// TwinCAT 3 PLC project MAIN
// ProgramVersion: 3.1.4026.24
// libraries:
//   Tc2_Standard, * (Beckhoff Automation GmbH)
//   Tc2_System, * (Beckhoff Automation GmbH)
// project tree:
//   DUTs/ E_AutoStep.TcDUT, E_HostCmdId.TcDUT, E_MachineState.TcDUT, ST_HostCmd.TcDUT, ST_PlcState.TcDUT
//   GVLs/ GVL_HMI.TcGVL
//   / PlcTask.TcTTO
//   POUs/ FB_AutoProcess.TcPOU, FB_HmiInterface.TcPOU, MAIN.TcPOU
// real-time tasks:
//   TASK PlcTask: cycle T#10ms, priority 20, ADS port 350

CONFIGURATION MAIN
    RESOURCE PLC ON TwinCAT3
        TASK PlcTask(INTERVAL := T#10ms, PRIORITY := 20);
        PROGRAM MAIN WITH PlcTask : MAIN;
    END_RESOURCE
END_CONFIGURATION

// ---- DUTs/E_AutoStep.TcDUT
TYPE E_AutoStep :
(
    Idle              := 0,
    CheckReady        := 10,
    TrayFeed          := 20,
    PickProduct       := 30,
    TopVisionAngle    := 40,
    RotateProduct     := 50,
    PlaceToRing       := 60,
    RingToClamp       := 70,
    ClampProduct      := 80,
    CoaxVision        := 90,
    CoaxAdjust        := 100,
    ScrewMove         := 110,
    ScrewTighten      := 120,
    RingReturn        := 130,
    PickBack          := 140,
    PlaceToTray       := 150,
    NextProduct       := 160,
    Finished          := 170,
    Error             := 999
);
END_TYPE

// ---- DUTs/E_HostCmdId.TcDUT
TYPE E_HostCmdId :
(
    None        := 0,
    StartAuto   := 1,
    Pause       := 2,
    ContinueRun := 3,
    Stop        := 4,
    Reset       := 5,
    ClearAlarm  := 6,
    HomeAll     := 7,
    ToManual    := 8,
    ToAuto      := 9,
    ManualAct   := 10
);
END_TYPE

// ---- DUTs/E_MachineState.TcDUT
TYPE E_MachineState :
(
    PowerOnCheck := 0,
    NeedHome     := 10,
    Homing       := 20,
    Standby      := 30,
    AutoRunning  := 40,
    Paused       := 50,
    Stopping     := 60,
    Alarm        := 70,
    Manual       := 80,
    Maintenance  := 90
);
END_TYPE

// ---- DUTs/ST_HostCmd.TcDUT
TYPE ST_HostCmd :
STRUCT
    Heartbeat       : UDINT;        // 上位机心跳
    CmdSeq          : UDINT;        // 命令序号，每发一次命令加 1
    CmdId           : E_HostCmdId;  // 命令编号
    RecipeId        : UINT;         // 配方号
    ManualStationId : UINT;         // 手动工位编号
    ManualActionId  : UINT;         // 手动动作编号
END_STRUCT
END_TYPE

// ---- DUTs/ST_PlcState.TcDUT
TYPE ST_PlcState :
STRUCT
    Heartbeat      : UDINT;           // PLC 心跳
    AckSeq         : UDINT;           // 已响应的命令序号
    MachineState   : E_MachineState;  // 设备总状态
    CurrentStep    : E_AutoStep;      // 当前自动工步
    AlarmCode      : UDINT;           // 当前报警代码

    AutoRunning    : BOOL;            // 自动运行中
    Paused         : BOOL;            // 暂停中
    AxisAllReady   : BOOL;            // 所有轴就绪
    EtherCATReady  : BOOL;            // EtherCAT 正常

    CurrentTray    : UINT;            // 当前料盘编号
    CurrentRow     : UINT;            // 当前行
    CurrentColumn  : UINT;            // 当前列

    GoodCount      : UDINT;           // OK 数量
    NgCount        : UDINT;           // NG 数量
    CycleTimeMs    : LREAL;           // 单件节拍
END_STRUCT
END_TYPE

// ---- GVLs/GVL_HMI.TcGVL
VAR_GLOBAL
    gHostCmd  : ST_HostCmd;   // 上位机写入
    gPlcState : ST_PlcState;  // PLC 返回上位机
END_VAR

// ---- POUs/MAIN.TcPOU
PROGRAM MAIN
VAR
    fbHmiInterface : FB_HmiInterface;
    fbAutoProcess  : FB_AutoProcess;
END_VAR

// 处理上位机命令
fbHmiInterface();

// 自动流程状态机
fbAutoProcess();

END_PROGRAM

// ---- POUs/FB_HmiInterface.TcPOU
FUNCTION_BLOCK FB_HmiInterface
VAR
    lastCmdSeq : UDINT := 0;
END_VAR

GVL_HMI.gPlcState.Heartbeat := GVL_HMI.gPlcState.Heartbeat + 1;

GVL_HMI.gPlcState.AxisAllReady := TRUE;
GVL_HMI.gPlcState.EtherCATReady := TRUE;

IF GVL_HMI.gPlcState.MachineState = 0 THEN
    GVL_HMI.gPlcState.MachineState := 30;
END_IF

IF GVL_HMI.gHostCmd.CmdSeq <> lastCmdSeq THEN

    lastCmdSeq := GVL_HMI.gHostCmd.CmdSeq;

    CASE GVL_HMI.gHostCmd.CmdId OF

        1:
            IF GVL_HMI.gPlcState.MachineState = 30 THEN
                GVL_HMI.gPlcState.MachineState := 40;
                GVL_HMI.gPlcState.AutoRunning := TRUE;
                GVL_HMI.gPlcState.Paused := FALSE;
                GVL_HMI.gPlcState.CurrentStep := 0;
            END_IF

        2:
            IF GVL_HMI.gPlcState.MachineState = 40 THEN
                GVL_HMI.gPlcState.MachineState := 50;
                GVL_HMI.gPlcState.AutoRunning := FALSE;
                GVL_HMI.gPlcState.Paused := TRUE;
            END_IF

        3:
            IF GVL_HMI.gPlcState.MachineState = 50 THEN
                GVL_HMI.gPlcState.MachineState := 40;
                GVL_HMI.gPlcState.AutoRunning := TRUE;
                GVL_HMI.gPlcState.Paused := FALSE;
            END_IF

        4:
            GVL_HMI.gPlcState.MachineState := 30;
            GVL_HMI.gPlcState.AutoRunning := FALSE;
            GVL_HMI.gPlcState.Paused := FALSE;
            GVL_HMI.gPlcState.CurrentStep := 0;

        5:
            GVL_HMI.gPlcState.AlarmCode := 0;
            GVL_HMI.gPlcState.MachineState := 30;
            GVL_HMI.gPlcState.AutoRunning := FALSE;
            GVL_HMI.gPlcState.Paused := FALSE;
            GVL_HMI.gPlcState.CurrentStep := 0;

        6:
            GVL_HMI.gPlcState.AlarmCode := 0;
            IF GVL_HMI.gPlcState.MachineState = 70 THEN
                GVL_HMI.gPlcState.MachineState := 30;
            END_IF

    END_CASE

    GVL_HMI.gPlcState.AckSeq := lastCmdSeq;

END_IF

END_FUNCTION_BLOCK

// ---- POUs/FB_AutoProcess.TcPOU
FUNCTION_BLOCK FB_AutoProcess
VAR
    stepTimer : TON;
    stepDelay : TIME := T#1S;
END_VAR

// 只有自动运行状态才推进流程
IF GVL_HMI.gPlcState.MachineState <> 40 THEN // AutoRunning
    stepTimer(IN := FALSE);
    RETURN;
END_IF

// 每一步延时 1 秒，方便上位机观察工步变化
stepTimer(IN := TRUE, PT := stepDelay);

IF NOT stepTimer.Q THEN
    RETURN;
END_IF

// 定时器到达后复位，准备下一步
stepTimer(IN := FALSE);

CASE GVL_HMI.gPlcState.CurrentStep OF

    0: // Idle
        GVL_HMI.gPlcState.CurrentStep := 10; // CheckReady

    10: // CheckReady
        IF GVL_HMI.gPlcState.AxisAllReady AND GVL_HMI.gPlcState.EtherCATReady THEN
            GVL_HMI.gPlcState.CurrentStep := 20; // TrayFeed
        ELSE
            GVL_HMI.gPlcState.AlarmCode := 1001;
            GVL_HMI.gPlcState.MachineState := 70; // Alarm
        END_IF

    20: // TrayFeed 料盘补给
        GVL_HMI.gPlcState.CurrentStep := 30; // PickProduct

    30: // PickProduct 三轴取料
        GVL_HMI.gPlcState.CurrentStep := 40; // TopVisionAngle

    40: // TopVisionAngle 角度相机识别
        GVL_HMI.gPlcState.CurrentStep := 50; // RotateProduct

    50: // RotateProduct 旋转夹爪校正角度
        GVL_HMI.gPlcState.CurrentStep := 60; // PlaceToRing

    60: // PlaceToRing 放入环形备料位
        GVL_HMI.gPlcState.CurrentStep := 70; // RingToClamp

    70: // RingToClamp 环形区旋转到夹紧位
        GVL_HMI.gPlcState.CurrentStep := 80; // ClampProduct

    80: // ClampProduct 夹紧产品
        GVL_HMI.gPlcState.CurrentStep := 90; // CoaxVision

    90: // CoaxVision 同轴度检测
        GVL_HMI.gPlcState.CurrentStep := 100; // CoaxAdjust

    100: // CoaxAdjust 同轴度调整
        GVL_HMI.gPlcState.CurrentStep := 110; // ScrewMove

    110: // ScrewMove 电批移动
        GVL_HMI.gPlcState.CurrentStep := 120; // ScrewTighten

    120: // ScrewTighten 拧紧螺钉
        GVL_HMI.gPlcState.CurrentStep := 130; // RingReturn

    130: // RingReturn 夹紧位旋回备料位
        GVL_HMI.gPlcState.CurrentStep := 140; // PickBack

    140: // PickBack 三轴取回产品
        GVL_HMI.gPlcState.CurrentStep := 150; // PlaceToTray

    150: // PlaceToTray 放回料盘
        GVL_HMI.gPlcState.GoodCount := GVL_HMI.gPlcState.GoodCount + 1;
        GVL_HMI.gPlcState.CurrentColumn := GVL_HMI.gPlcState.CurrentColumn + 1;
        GVL_HMI.gPlcState.CurrentStep := 160; // NextProduct

    160: // NextProduct 下一个产品
        IF GVL_HMI.gPlcState.CurrentColumn >= 6 THEN
            GVL_HMI.gPlcState.CurrentColumn := 0;
            GVL_HMI.gPlcState.CurrentRow := GVL_HMI.gPlcState.CurrentRow + 1;
        END_IF

        IF GVL_HMI.gPlcState.CurrentRow >= 4 THEN
            GVL_HMI.gPlcState.CurrentRow := 0;
            GVL_HMI.gPlcState.CurrentTray := GVL_HMI.gPlcState.CurrentTray + 1;
        END_IF

        IF GVL_HMI.gPlcState.CurrentTray >= 5 THEN
            GVL_HMI.gPlcState.CurrentStep := 170; // Finished
        ELSE
            GVL_HMI.gPlcState.CurrentStep := 20; // 回到料盘补给/下一件流程
        END_IF

    170: // Finished 全部完成
        GVL_HMI.gPlcState.AutoRunning := FALSE;
        GVL_HMI.gPlcState.MachineState := 30; // Standby
        GVL_HMI.gPlcState.CurrentStep := 0;   // Idle

ELSE
    GVL_HMI.gPlcState.AlarmCode := 9999;
    GVL_HMI.gPlcState.MachineState := 70; // Alarm

END_CASE

END_FUNCTION_BLOCK
